// TIA Portal V17 export
// export: Created 2025-03-10T13:11:50.9981203Z, ExportSetting WithDefaults, DisplayName Totally Integrated Automation Portal, DisplayVersion V17 Update 8, DisplayName TIA Portal Openness, DisplayVersion V17 Update 8, DisplayName TIA Portal Version Control Interface, DisplayVersion V17, DisplayName SINAMICS Startdrive Advanced, DisplayVersion V17 SP2, DisplayName SINAMICS Startdrive G110M, G120, G120C, G120D, G120P, G115D, DisplayVersion V17 SP2, DisplayName SINAMICS Startdrive G130, G150, S120, S150, SINAMICS MV, S210, DisplayVersion V17 SP2, DisplayName STEP 7 Professional, DisplayVersion V17 Update 8, DisplayName SINUMERIK ONE STEP 7 Toolbox, DisplayVersion V17 Update 12, DisplayName SINUMERIK 840D sl STEP 7 Toolbox, DisplayVersion V17 Update 12, DisplayName STEP 7 Safety, DisplayVersion V17 Update 6, DisplayName WinCC Advanced, DisplayVersion V17 Update 8
VAR_GLOBAL   // PLC tag table "TAGS_IO_OTHER_CLADDING"
   "/////_UNIT_01_STATION_3_PYROMETER_/////" AT %M1300.0 : Bool;   // /////_UNIT_01_STATION_3_PYROMETER/////
   "/////_UNIT_01_PART_PRESENT_CONTROL_/////" AT %M1300.2 : Bool;   // /////_UNIT_01_PART_PRESENT_CONTROL/////
   "/////_UNIT_01_JAW_CHUCK_GRIPPER_CONTROL/////" AT %M1300.4 : Bool;   // /////_UNIT_01_JAW_CHUCK_GRIPPER_CONTROL/////
   "/////_U01_PT100_TEMPERATURE_SENSORS_/////" AT %M1300.6 : Bool;   // /////_U01_PT100_TEMPERATURE_SENSORS_*/////
   U01_KF730_SENSOR_1 AT %MW1301 : Int;   // UNIT 01 KF730 SENSOR 1
   U01_KF730_SENSOR_2 AT %MW1303 : Int;   // UNIT 01 KF730 SENSOR 2
   U01_KF730_SENSOR_3 AT %MW1305 : Int;   // UNIT 01 KF730 SENSOR 3
   U01_KF730_SENSOR_4 AT %MW1307 : Int;   // UNIT 01 KF730 SENSOR 4
   U01_KF730_SENSOR_5 AT %MW1309 : Int;   // UNIT 01 KF730 SENSOR 5
   U01_KF730_SENSOR_6 AT %MW1311 : Int;   // UNIT 01 KF730 SENSOR 6
   U01_PT100_400_SENSOR_1 AT %MW1313 : Int;   // UNIT 01 PT100 400 SENSOR 1
   U01_PT100_400_SENSOR_2 AT %MW1315 : Int;   // UNIT 01 PT100 400 SENSOR 2
   U01_PT100_400_SENSOR_3 AT %MW1317 : Int;   // UNIT 01 PT100 400 SENSOR 3
   U01_PT100_400_SENSOR_4 AT %MW1319 : Int;   // UNIT 01 PT100 400 SENSOR 4
   U01_PT100_ENVIROMENT_1 AT %MW1321 : Int;   // UNIT 01 ENVIROMENT PT100 1
   U01_PT100_ENVIROMENT_2 AT %MW1323 : Int;   // UNIT 01 ENVIROMENT PT100 2
   U01_IN_POSITION AT %I500.6 : Bool;   // U01 READY TO MOVE. BOLT OK
   U01_TURN_CONTROL_FIXT AT %IW518 : Word;   // UNIT 01 FIXTURE TURNING CONTROL
   U01_AXIS_X13_ADVANCED_POS AT %I570.0 : Bool;   // AXIS X13 ADVANCED POSITION INPUT
   U01_AXIS_X13_GARAGE_POS AT %I570.1 : Bool;   // AXIS X13 GARAGE POSITION INPUT
   U01_AXIS_X13_RETURNED_POS AT %I570.2 : Bool;   // AXIS X13 RETURNED POSITION INPUT
   U01_AXIS_Z13_DOWN_POS AT %I570.3 : Bool;   // AXIS Z13 DOWN POSITION INPUT
   U01_AXIS_Z13_UP_POS AT %I570.4 : Bool;   // AXIS Z13 UP POSITION INPUT
   U01_AXIS_Z13_GARAGE_POS AT %I570.7 : Bool;   // AXIS Z13 GARAGE POSITION INPUT
   U01_STA_3_PRESSURE AT %IW526 : Word;   // UNIT 01 STATION 3 PRESSURE
   U01_LASER_COOLING_NOZZLE_FLOW_SP AT %I70.1 : Bool;   // UNIT 01 LASER COOLING NOZZLE FLOW SENSOR SETPOINT
   U01_LASER_COOLING_NOZZLE_TEMP_SP AT %I71.1 : Bool;   // UNIT 01 LASER COOLING NOZZLE TEMPERATURE SENSOR SETPOINT
   U01_LASER_COOLING_HEAD_FLOW_SP AT %I70.2 : Bool;   // UNIT 01 LASER COOLING HEAD FLOW SENSOR SETPOINT
   U01_LASER_COOLING_HEAD_TEMP_SP AT %I71.2 : Bool;   // UNIT 01 LASER COOLING HEAD TEMPERATURE SENSOR SETPOINT
   U01_LASER_COOLING_OUTPUT_FLOW_VALUE AT %MW1335 : Int;   // UNIT 01 LASER COOLING OUTPUT FLOW SENSOR VALUE
   U01_LASER_COOLING_OUTPUT_TEMP_VALUE AT %MW1337 : Word;   // UNIT 01 LASER COOLING OUTPUT TEMPERATURE SENSOR VALUE
   U01_LASER_COOLING_OUTPUT_FLOW_SP AT %I70.0 : Bool;   // UNIT 01 LASER COOLING OUTPUT FLOW SENSOR SETPOINT
   U01_LASER_COOLING_OUTPUT_TEMP_SP AT %I71.0 : Bool;   // UNIT 01 LASER COOLING OUTPUT TEMPERATURE SENSOR SETPOINT
   "/////_UNIT_02_STATION_3_PYROMETER/////" AT %M1338.0 : Bool;   // /////_UNIT_02_STATION_3_PYROMETER/////
   "/////_UNIT_02_PART_PRESENT_CONTROL/////" AT %M1338.2 : Bool;   // /////_UNIT_02_PART_PRESENT_CONTROL/////
   "/////_UNIT_02_JAW_CHUCK_GRIPPER_CONTROL/////" AT %M1338.4 : Bool;   // /////_UNIT_02_JAW_CHUCK_GRIPPER_CONTROL/////
   "/////_U02_PT100_TEMPERATURE_SENSORS_/////" AT %M1338.6 : Bool;   // /////_U02_PT100_TEMPERATURE_SENSORS_*/////
   U02_KF730_SENSOR_1 AT %MW1339 : Int;   // UNIT 02 KF730 SENSOR 1
   U02_KF730_SENSOR_2 AT %MW1341 : Int;   // UNIT 02 KF730 SENSOR 2
   U02_KF730_SENSOR_3 AT %MW1343 : Int;   // UNIT 02 KF730 SENSOR 3
   U02_KF730_SENSOR_4 AT %MW1345 : Int;   // UNIT 02 KF730 SENSOR 4
   U02_KF730_SENSOR_5 AT %MW1347 : Int;   // UNIT 02 KF730 SENSOR 5
   U02_KF730_SENSOR_6 AT %MW1349 : Int;   // UNIT 02 KF730 SENSOR 6
   U02_PT100_400_SENSOR_1 AT %MW1351 : Int;   // UNIT 02 PT100 400 SENSOR 1
   U02_PT100_400_SENSOR_2 AT %MW1353 : Int;   // UNIT 02 PT100 400 SENSOR 2
   U02_PT100_400_SENSOR_3 AT %MW1355 : Int;   // UNIT 02 PT100 400 SENSOR 3
   U02_PT100_400_SENSOR_4 AT %MW1357 : Int;   // UNIT 02 PT100 400 SENSOR 4
   U02_PT100_ENVIROMENT_1 AT %MW1359 : Int;   // UNIT 02 ENVIROMENT PT100 1
   U02_PT100_ENVIROMENT_2 AT %MW1361 : Int;   // UNIT 02 ENVIROMENT PT100 2
   "/////_UNIT_02_OTHERS_/////" AT %M1363.0 : Bool;   // /////_UNIT_02_OTHERS_/////
   U02_IN_POSITION AT %I1500.6 : Bool;   // U02 READY TO MOVE. BOLT OK
   U02_TURN_CONTROL_FIXT AT %IW1518 : Word;   // UNIT 01 FIXTURE TURNING CONTROL
   U02_X23_ADVANCED_POS AT %I1570.0 : Bool;   // AXIS X23 ADVANCED POSITION INPUT
   U02_X23_GARAGE_POS AT %I1570.1 : Bool;   // AXIS X23 GARAGE POSITION INPUT
   U02_X23_RETURNED_POS AT %I1570.2 : Bool;   // AXIS X23 RETURNED POSITION INPUT
   U02_Z23_DOWN_POS AT %I1570.3 : Bool;   // AXIS Z23 DOWN POSITION INPUT
   U02_Z23_UP_POS AT %I1570.4 : Bool;   // AXIS Z23 UP POSITION INPUT
   U02_Z23_GARAGE_POS AT %I1570.7 : Bool;   // AXIS Z23 GARAGE POSITION INPUT
   U02_LASER_COOLING_NOZZLE_FLOW_SP AT %I1070.1 : Bool;   // UNIT 01 LASER COOLING NOZZLE FLOW SENSOR SETPOINT
   U01_STA_1_PUSHER_W11_RTND AT %I470.1 : Bool;   // UNIT 01 PUSHER RETURNED
   U01_FIX_GRIPPER_CONTROL AT %IW468 : Word;   // UNIT 01 FIXTURE GRIPPER/JAW CHUCK CONTROL
   U02_FIX_GRIPPER_CONTROL AT %IW1468 : Word;   // UNIT 02 FIXTURE GRIPPER/JAW CHUCK CONTROL
   U02_STA_1_PUSHER_W21_RTND AT %I1470.1 : Bool;   // UNIT 02 PUSHER RETURNED
   "/////_UNIT_01_OTHERS_/////" AT %M1325.0 : Bool;   // /////_UNIT_01_OTHERS_/////
   U02_LASER_COOLING_NOZZLE_TEMP_VALUE AT %IW1652 : Int;   // UNIT 02 LASER COOLING NOZZLE TEMP VALUE
   U01_LASER_COOLING_NOZZLE_FLOW_VALUE AT %IW650 : Int;   // UNIT 01 LASER COOLING NOZZLE FLOW VALUE
   U02_LASER_COOLING_HEAD_TEMP_VALUE AT %ID1664 : DInt;   // UNIT 02 LASER COOLING HEAD TEMP VALUE
   U01_LASER_COOLING_HEAD_TEMP_VALUE AT %ID664 : DInt;   // UNIT 01 LASER COOLING HEAD TEMPERATURE VALUE
   U02_LASER_COOLING_NOZZLE_FLOW_VALUE AT %IW1650 : Int;   // UNIT 02 LASER COOLING NOZZLE FLOW VALUE
   U01_LASER_COOLING_NOZZLE_TEMP_VALUE AT %IW652 : Int;   // UNIT 01 LASER COOLING NOZZLE TEMPERATURE VALUE
   U02_LASER_COOLING_HEAD_FLOW_VALUE AT %ID1658 : DInt;   // UNIT 02 LASER COOLING HEAD FLOW VALUE
   U01_LASER_COOLING_HEAD_FLOW_VALUE AT %ID658 : DInt;   // UNIT 01 LASER COOLING HEAD FLOW VALUE
   U02_STA3_CLEANING_VALVE AT %Q68.0 : Bool;
   U01_STA3_CLEANING_VALVE AT %Q1068.0 : Bool;
   U01_TURCK_LD_PART_Q AT %Q606.3 : Bool;   // UNIT 01 BIMANUAL LOADED PART OUTPUT
   U01_TURCK_UNLD_PART_Q AT %Q606.1 : Bool;   // UNIT 01 BIMANUAL UNLOADED PART OUTPUT
   U01_TURCK_RESET_FAULTS_I AT %I606.4 : Bool;   // UNIT 01 BIMANUAL RESET FAULTS INPUT
   U01_TURCK_START_CYCLE_Q AT %Q606.7 : Bool;   // UNIT 01 BIMANUAL START CYCLE OUTPUT
   U01_TURCK_UNLD_PART_I AT %I606.0 : Bool;   // UNIT 01 BIMANUAL UNLOAD PART INPUT
   U01_TURCK_RESET_FAULTS_Q AT %Q606.5 : Bool;   // UNIT 01 BIMANUAL RESET FAULTS OUTPUT
   U01_TURCK_LD_PART_I AT %I606.2 : Bool;   // UNIT 01 BIMANUAL LOAD PART INPUT
   U01_TURCK_START_CYCLE_I AT %I606.6 : Bool;   // UNIT 01 BIMANUAL START CYCLE INPUT
   U01_PYRO_CURRENT_TRANSMISSION AT %ID3644 : Real;   // UNIT 01 PYROMETER CURRENT TRANSMISSION
   U01_PYRO_HEAD_TEMPERATURE AT %ID3608 : Real;   // UNIT 01 PYROMETER HEAD TEMPERATURE
   U02_PYRO_CURRENT_TRANSMISSION AT %ID3744 : Real;   // UNIT 02 PYROMETER CURRENT TRANSMISSION
   U02_PYRO_HEAD_TEMPERATURE AT %ID3708 : Real;   // UNIT 02 PYROMETER HEAD TEMPERATURE
   U01_PYRO_PROCESS_TEMPERATURE AT %ID3604 : Real;   // UNIT 01 PYROMETER PROCESS TEMPERATURE
   U01_PYRO_T2_TEMPERATURE AT %ID3632 : Real;   // UNIT 01 PYROMETER T2 TEMPERATURE
   U02_PYRO_PROCESS_TEMPERATURE AT %ID3704 : Real;   // UNIT 02 PYROMETER PROCESS TEMPERATURE
   U02_PYRO_CURRENT_EMISSIVITY AT %ID3740 : Real;   // UNIT 02 PYROMETER CURRENT EMISSIVITY
   U01_PYRO_CURRENT_EMISSIVITY AT %ID3640 : Real;   // UNIT 01 PYROMETER CURRENT EMISSIVITY
   U01_PYRO_T1_TEMPERATURE AT %ID3628 : Real;   // UNIT 01 PYROMETER T1 TEMPERATURE
   U01_PYRO_DEVICE_STATUS AT %ID3600 : Real;   // UNIT 01 PYROMETER DEVICE STATUS
   U02_PYRO_DEVICE_STATUS AT %ID3700 : Real;   // UNIT 02 PYROMETER DEVICE STATUS
   U02_PYRO_T1_TEMPERATURE AT %ID3728 : Real;   // UNIT 02 PYROMETER T1 TEMPERATURE
   U02_PYRO_T2_TEMPERATURE AT %ID3732 : Real;   // UNIT 02 PYROMETER T2 TEMPERATURE
   U02_LASER_COOLING_HEAD_TEMP_SP AT %I1071.2 : Bool;   // UNIT 02 LASER COOLING HEAD TEMPERATURE SENSOR SETPOINT
   U02_LASER_COOLING_NOZZLE_TEMP_SP AT %I1071.1 : Bool;   // UNIT 02 LASER COOLING NOZZLE TEMPERATURE SENSOR SETPOINT
   U02_LASER_COOLING_OUTPUT_FLOW_VALUE AT %MW1374 : Int;   // UNIT 02 LASER COOLING OUTPUT FLOW SENSOR VALUE
   U02_LASER_COOLING_HEAD_FLOW_SP AT %I1070.2 : Bool;   // UNIT 02 LASER COOLING HEAD FLOW SENSOR SETPOINT
   U02_LASER_COOLING_OUTPUT_FLOW_SP AT %I1070.0 : Bool;   // UNIT 02 LASER COOLING OUTPUT FLOW SENSOR SETPOINT
   U02_LASER_COOLING_OUTPUT_TEMP_VALUE AT %MW1376 : Word;   // UNIT 02 LASER COOLING OUTPUT TEMPERATURE SENSOR VALUE
   U02_LASER_COOLING_OUTPUT_TEMP_SP AT %I1071.0 : Bool;   // UNIT 02 LASER COOLING OUTPUT TEMPERATURE SENSOR SETPOINT
   U01_KF320_400_PT100_1 AT %IW512 : Int;   // UNIT 01 KF320 400ºC PT100 SENSOR 1
   U02_KF1320_400_PT100_2 AT %IW1516 : Int;   // UNIT 02 KF1320 400ºC PT100 SENSOR 2
   U01_KF320_400_PT100_2 AT %IW516 : Int;   // UNIT 01 KF320 400ºC PT100 SENSOR 2
   U02_KF1320_400_PT100_1 AT %IW1512 : Int;   // UNIT 02 KF1320 400ºC PT100 SENSOR 1
   U01_SHIELD_COOLING_FLOW_VALUE AT %IW690 : Int;   // UNIT 01 SHIELD COOLING FLOW VALUE
   U02_SHIELD_COOLING_TEMP_VALUE AT %IW1692 : Int;   // UNIT 02 SHIELD COOLING TEMPERATURE VALUE
   U01_SHIELD_COOLING_TEMP_VALUE AT %IW692 : Int;   // UNIT 01 SHIELD COOLING TEMPERATURE VALUE
   U02_SHIELD_COOLING_FLOW_VALUE AT %IW1690 : Int;   // UNIT 02 SHIELD COOLING FLOW VALUE
   U02_STA_3_PRESSURE AT %IW1526 : Word;   // UNIT 02 STATION 3 PRESSURE
END_VAR
